(* CoDeSys 2.3.9.41 project: plc_110_main.pro *)
(* Libraries: D:\Projects\LittleProjects\Physical\Apartments\Slavutich2\SmartHouse\CoDeSys\lib\Timer.lib 12.1.22 22:29:23, STANDARD.LIB 4.10.05 11:14:46, IECSFC.LIB 13.4.06 15:51:28, C:\Program Files (x86)\Common Files\CAA-Targets\3S\Lib_PLCWinNT\SysLibCallback.lib 26.9.08 16:43:52, ANALYZATION.LIB 5.10.99 09:05:06 *)

(* PLC configuration (modules and I/O channels)
U1_FDI1_dimmer_button AT %IX0.0 [BitInput] FDI1_dimmer_button {ChannellName = Enter name}
U1_FDI2_dimmer_up AT %IX0.1 [BitInput] FDI2_dimmer_up {ChannellName = Enter name}
U1_FDI3_dimmer_down AT %IX0.2 [BitInput] FDI3_dimmer_down {ChannellName = Enter name}
U1_FDI4_NC AT %IX0.3 [BitInput] FDI4_NC {ChannellName = Enter name}
AT %IB1.0 [ByteInput] 8 discrete inputs {ChannellName = Enter name}
AT %IB1.1 [ByteInput] 8 discrete inputs {ChannellName = Enter name}
AT %IB1.2 [ByteInput] 8 discrete inputs {ChannellName = Enter name}
AT %IB1.3 [ByteInput] 8 discrete inputs {ChannellName = Enter name}
U1_DO1_warm_floor_room AT %QX2.0 [BitOutput] DO1_warm_floor_room {ChannellName = Enter name}
U1_DO2_warm_floor_logia AT %QX2.1 [BitOutput] DO2_warm_floor_logia {ChannellName = Enter name}
U1_DO3_warm_floor_kitchen AT %QX2.2 [BitOutput] DO3_warm_floor_kitchen {ChannellName = Enter name}
U1_DO4_warm_floor_hall AT %QX2.3 [BitOutput] DO4_warm_floor_hall {ChannellName = Enter name}
AT %QB3.0 [ByteOutput] 8 discrete outputs {ChannellName = Enter name}
AT %QB3.1 [ByteOutput] 8 discrete outputs {ChannellName = Enter name}
AT %QB3.2 [ByteOutput] 4 discrete outputs {ChannellName = Enter name}
Special input [ID103] node 4, in %IB4 out %QB4 {ChannellName = Special input}
  AT %IX4.0 [BitInput] Special input {ChannellName = Enter name}
Special output [ID104] node 5, in %IB5 out %QB5 {ChannellName = Special output}
  U1_PLC_speaker AT %QX5.0 [BitOutput] PLC_speaker {ChannellName = Enter name}
AT %QD6.0 [DWordOutput] Last address {ChannellName = Enter name}
AT %QW6.1 [WordOutput] Last error {ChannellName = Enter name}
RS-485-1 [COM1_USART] node 0, in %IB6.0 out %QB6.0 {ChannellName = RS-485-1; CommunicationSpeed = 115200; Parity = NO PARITY CHECK; BitLength = 8 bits; StopLength = One stop bit; InterfaceType = RS485; FrameOriented = RTU; Timeout = 0; Visibility = No}
Universal Modbus device [ID2000] node 1, in %IB6.1 out %QB6.1 {ChannellName = M1; ModuleIP = 10:0:0:223; ServiceTimeout = 150; TCPport = 502; NetMode = Serial; ModuleSlaveAddress = 1; RequestType = Both; PeriodOfService = 1000; Visibility = No; RepeatCounter = 0; ByteSequence = Trace_mode}
  AT %QB6.1.0 [ComChannel] Command (0xff - Start) {ChannellName = Enter name}
M1_DO1_door_lock_on AT %QW6.1.0.0 [WordOutput] {ChannellName = Enter name}
M1_DO2_doorbell_on AT %QW6.1.1.0 [WordOutput] {ChannellName = Enter name}
M1_DO3_door_lock_open_close AT %QW6.1.2.0 [WordOutput] {ChannellName = Enter name}
M1_DO4_cold_water_valve_close AT %QW6.1.3.0 [WordOutput] {ChannellName = Enter name}
M1_DO5_hot_water_valve_close AT %QW6.1.4.0 [WordOutput] {ChannellName = Enter name}
M1_DO6_water_valves_on AT %QW6.1.5.0 [WordOutput] {ChannellName = Enter name}
M1_DO7_NC AT %QW6.1.6.0 [WordOutput] {ChannellName = Enter name}
M1_DO8_siren_on AT %QW6.1.7.0 [WordOutput] {ChannellName = Enter name}
M1_DO_state AT %QW6.1.8.0 [WordOutput] {ChannellName = Enter name}
Universal Modbus device [ID2000] node 2, in %IB6.2 out %QB6.2 {ChannellName = Universal Modbus device; ModuleIP = 10:0:0:223; ServiceTimeout = 150; TCPport = 502; NetMode = Serial; ModuleSlaveAddress = 2; RequestType = Both; PeriodOfService = 1000; Visibility = No; RepeatCounter = 0; ByteSequence = Trace_mode}
  AT %QB6.2.0 [ComChannel] Command (0xff - Start) {ChannellName = Enter name}
M2_DO1_room_jalousie_up_down AT %QW6.2.0.0 [WordOutput] {ChannellName = Enter name}
M2_DO2_room_jalousie_on AT %QW6.2.1.0 [WordOutput] {ChannellName = Enter name}
M2_DO3_logia_jalousie_up_down AT %QW6.2.2.0 [WordOutput] {ChannellName = Enter name}
M2_DO4_logia_jalousie_on AT %QW6.2.3.0 [WordOutput] {ChannellName = Enter name}
M2_DO5_batroom_ventilation_fast_slow AT %QW6.2.4.0 [WordOutput] {ChannellName = Enter name}
M2_DO6_batroom_ventilation_on AT %QW6.2.5.0 [WordOutput] {ChannellName = Enter name}
M2_DO7_room_ventilation_fast_slow AT %QW6.2.6.0 [WordOutput] {ChannellName = Enter name}
M2_DO8_room_ventilation_on AT %QW6.2.7.0 [WordOutput] {ChannellName = Enter name}
M2_DO_state AT %QW6.2.8.0 [WordOutput] {ChannellName = Enter name}
AT %QB6.3.0 [ComChannel] Command (0xff - Start) {ChannellName = Enter name}
M3_IN1_status_warm_floor_room AT %QW6.3.0.0 [WordOutput] {ChannellName = Enter name}
M3_IN1_time_warm_floor_room AT %QW6.3.1.0 [WordOutput] {ChannellName = Enter name}
M3_IN1_temper_warm_floor_room AT %QD6.3.2.0 [FloatOutput] {ChannellName = Enter name}
M3_IN2_status_warm_floor_logia AT %QW6.3.3.0 [WordOutput] {ChannellName = Enter name}
M3_IN2_time_warm_floor_logia AT %QW6.3.4.0 [WordOutput] {ChannellName = Enter name}
M3_IN2_temper_warm_floor_logia AT %QD6.3.5.0 [FloatOutput] {ChannellName = Enter name}
M3_IN3_status_warm_floor_kitchen AT %QW6.3.6.0 [WordOutput] {ChannellName = Enter name}
M3_IN3_time_warm_floor_kitchen AT %QW6.3.7.0 [WordOutput] {ChannellName = Enter name}
M3_IN3_temper_warm_floor_kitchen AT %QD6.3.8.0 [FloatOutput] {ChannellName = Enter name}
M3_IN4_status_warm_floor_hall AT %QW6.3.9.0 [WordOutput] {ChannellName = Enter name}
M3_IN4_time_warm_floor_hall AT %QW6.3.10.0 [WordOutput] {ChannellName = Enter name}
M3_IN4_temper_warm_floor_hall AT %QD6.3.11.0 [FloatOutput] {ChannellName = Enter name}
M3_IN5_status_warm_floor_bathroom AT %QW6.3.12.0 [WordOutput] {ChannellName = Enter name}
M3_IN5_time_warm_floor_bathroom AT %QW6.3.13.0 [WordOutput] {ChannellName = Enter name}
M3_IN5_temper_warm_floor_bathroom AT %QD6.3.14.0 [FloatOutput] {ChannellName = Enter name}
M3_IN6_status_outdoor AT %QW6.3.15.0 [WordOutput] {ChannellName = Enter name}
ID2003NoNoINTRegister input module AT %QW6.3.16.0 [WordOutput] B%QB%MB%MM3_IN6_time_outdoor {ChannellName = Enter name}
M3_IN6_temper_outdoor AT %QD6.3.17.0 [FloatOutput] {ChannellName = Enter name}
M3_IN7_status_box AT %QW6.3.18.0 [WordOutput] {ChannellName = Enter name}
M3_IN7_time_box AT %QW6.3.19.0 [WordOutput] {ChannellName = Enter name}
M3_IN7_temper_box AT %QD6.3.20.0 [FloatOutput] {ChannellName = Enter name}
M3_IN8_status_luminosity_room AT %QW6.3.21.0 [WordOutput] {ChannellName = Enter name}
M3_IN8_time_luminosity_room AT %QW6.3.22.0 [WordOutput] {ChannellName = Enter name}
M3_IN8_luminosity_room AT %QD6.3.46.0 [FloatOutput] {ChannellName = Enter name}
AT %QB6.4.0 [ComChannel] Command (0xff - Start) {ChannellName = Enter name}
M4_AO1_room_converter_speed AT %QW6.4.0.0 [WordOutput] {ChannellName = Enter name}
M4_AO2_logia_converter_speed AT %QW6.4.1.0 [WordOutput] {ChannellName = Enter name}
M4_AO_3_NC AT %QW6.4.2.0 [WordOutput] {ChannellName = Enter name}
M4_AO_4_NC AT %QW6.4.3.0 [WordOutput] {ChannellName = Enter name}
M4_AO_5_NC AT %QW6.4.4.0 [WordOutput] {ChannellName = Enter name}
M4_AO_6_NC AT %QW6.4.5.0 [WordOutput] {ChannellName = Enter name}
AT %QB6.5.0 [ComChannel] Command (0xff - Start) {ChannellName = Enter name}
M5_AO1_room_light_1 AT %QW6.5.0.0 [WordOutput] {ChannellName = Enter name}
M5_AO2_room_light_2 AT %QW6.5.1.0 [WordOutput] {ChannellName = Enter name}
M5_AO3_logia_light AT %QW6.5.2.0 [WordOutput] {ChannellName = Enter name}
M5_AO4_kitchen_light AT %QW6.5.3.0 [WordOutput] {ChannellName = Enter name}
M5_AO5_hall_light AT %QW6.5.4.0 [WordOutput] {ChannellName = Enter name}
M5_AO6_bathroom_light AT %QW6.5.5.0 [WordOutput] {ChannellName = Enter name}
TCP [TCP_ID221] node 0, in %IB7.0.0 out %QB7.0.0 {ChannellName = TCP; RemotePort = 502; Visibility = No}
8 bits [8Bit] node 1, in %IB7.1 out %QB7.1 {ChannellName = 8 bit}
  AT %QB7.1.0 [ByteOutput] {ChannellName = Enter name}
8 bits [8Bit] node 2, in %IB7.2 out %QB7.2 {ChannellName = 8 bit}
  AT %QB7.2.0 [ByteOutput] {ChannellName = Enter name}
  AT %QB7.3.0 [ByteOutput] {ChannellName = Enter name}
  AT %QB7.4.0 [ByteOutput] {ChannellName = Enter name}
U1_R_002_room_light_intensity_1 AT %QW7.5.0 [WordOutput] {ChannellName = Enter name}
U1_R_003_room_light_intensity_2 AT %QW7.6.0 [WordOutput] {ChannellName = Enter name}
U1_R_004_logia_light_intensity AT %QW7.7.0 [WordOutput] {ChannellName = Enter name}
U1_R_005_kitchen_light_intensity AT %QW7.8.0 [WordOutput] {ChannellName = Enter name}
U1_R_006_hall_light_intensity AT %QW7.9.0 [WordOutput] {ChannellName = Enter name}
U1_R_007_bathroom_light_intensity AT %QW7.10.0 [WordOutput] {ChannellName = Enter name}
U1_R_008_room_light_change_rate AT %QW7.11.0 [WordOutput] {ChannellName = Enter name}
U1_R_009_other_light_change_rate AT %QW7.12.0 [WordOutput] {ChannellName = Enter name}
U1_R_010_room_light_correction_in_auto AT %QW7.13.0 [WordOutput] {ChannellName = Enter name}
*)

(* Task configuration *)
TASK U1_FDI1_dimmer_button (PRIORITY := 1, SINGLE := U1_FDI1_dimmer_button);
	DIMMER_HANDLER(act:=1);
END_TASK
TASK U1_FDI2_dimmer_up (PRIORITY := 1, SINGLE := U1_FDI2_dimmer_up);
	DIMMER_HANDLER(act:=2);
END_TASK
TASK FDI3_dimmer_down (PRIORITY := 1, SINGLE := U1_FDI3_dimmer_down);
	DIMMER_HANDLER(act:=3);
END_TASK
TASK dimmer_handler_tick (PRIORITY := 1, INTERVAL := T#100ms);
	DIMMER_HANDLER(act:=0);
END_TASK
TASK switch_handler_tick (PRIORITY := 1, INTERVAL := T#50ms);
	SWITCH_HANDLER();
END_TASK
TASK light_driver_tick (PRIORITY := 1, INTERVAL := T#40ms);
	LIGHT_DRIVER();
END_TASK
TASK light_auto_control_tick (PRIORITY := 1, INTERVAL := T#100ms);
	LIGHT_AUTO_CONTROL();
END_TASK

(* Global variable list: Global_Variables *)
VAR_GLOBAL
    PLC_STATUS: INT := 0;
END_VAR
VAR_GLOBAL CONSTANT
	PLC_RUN: INT := 2;
END_VAR

(* POU DIMMER_HANDLER, ST *)
PROGRAM DIMMER_HANDLER
VAR_INPUT
    act: INT; (* Action: 0 - tick (each 100 mills), 1 - U1_FDI1_dimmer_button, 2 - U1_FDI2_dimmer_up, 3 - FDI3_dimmer_down *)
END_VAR

VAR CONSTANT
    (* Input actions *)
    TICK: INT := 0;
    DIMMER_BUTTON: INT := 1;
    DIMMER_UP: INT := 2;
    DIMMER_DOWN: INT := 3;

    (* Parameters *)
    INDICATOR_BLINCK_TIME: INT := 3; (* 300 mills *)
    NUM_BLINCK_TO_SWITCH_MODE: INT := 4;  (* (300 * 4 * 2)mills *)
    DIMMER_RESET_TIME: INT := 100; (* 10 seconds *)
    DIMMING_STEP: INT := 10;
    DIMMING_MAX_VALUE: INT := 1000;
    ROOM_LIGHT_CHANGE_RATE: INT := 2;
    OTHER_LIGHT_CHANGE_RATE: INT := 5;
END_VAR

VAR
    dimmer_swith_count: INT := -1;
    dimmer_reset_count: INT := 0;
    is_room_dimmer: BOOL := TRUE;
    count: INT := 0;
END_VAR
(*
    Handeling of dimmer control handle

    Author: CAB 
    Cseated: 2022.01.25
*)

IF PLC_STATUS = PLC_RUN THEN
    IF act = TICK THEN
        IF U1_FDI1_dimmer_button AND dimmer_swith_count < (INDICATOR_BLINCK_TIME * NUM_BLINCK_TO_SWITCH_MODE * 2) AND dimmer_swith_count >= 0 THEN
            (* Count until switch dimmer mode room/other *)
            U1_DO12_dimer_mode_indication := ((dimmer_swith_count / INDICATOR_BLINCK_TIME) MOD 2) = BOOL_TO_INT(NOT is_room_dimmer);
            dimmer_swith_count := dimmer_swith_count + 1;

        ELSIF U1_FDI1_dimmer_button AND dimmer_swith_count > 0 THEN
            (* Do switch dimmer mode room/other   *)
            is_room_dimmer := NOT is_room_dimmer;
            U1_DO12_dimer_mode_indication := NOT is_room_dimmer;
            dimmer_swith_count := -1;

        ELSIF (NOT U1_FDI1_dimmer_button) AND dimmer_swith_count > 0 THEN
            (* Set mode indicator in case dimmer button is off before mode switched*)
            U1_DO12_dimer_mode_indication := NOT is_room_dimmer;
            dimmer_swith_count := -1;
        END_IF

        IF NOT is_room_dimmer THEN
            IF dimmer_reset_count >= DIMMER_RESET_TIME THEN
                is_room_dimmer := TRUE;
                U1_DO12_dimer_mode_indication := FALSE;
            END_IF
            dimmer_reset_count := dimmer_reset_count + 1;
        END_IF

    ELSIF act = DIMMER_BUTTON THEN
        U1_DO12_dimer_mode_indication := is_room_dimmer;
        dimmer_swith_count := 0;
        dimmer_reset_count := 0;
        U1_C_024_room_light_auto := FALSE; (* Reset light auto controll *)

    ELSIF act = DIMMER_UP THEN
        IF U1_FDI3_dimmer_down THEN
            IF is_room_dimmer AND NOT U1_C_024_room_light_auto THEN
                (* Decrising of room dimmers *)

                IF U1_C_016_room_light_1_on OR U1_C_017_room_light_2_on THEN
                    U1_R_008_room_light_change_rate := ROOM_LIGHT_CHANGE_RATE;
                END_IF

                IF U1_C_016_room_light_1_on AND U1_R_002_room_light_intensity_1 > DIMMING_STEP THEN
                    U1_R_002_room_light_intensity_1 := U1_R_002_room_light_intensity_1 - DIMMING_STEP;
                ELSIF U1_C_016_room_light_1_on THEN
                    U1_R_002_room_light_intensity_1 := 0;
                END_IF

                IF U1_C_017_room_light_2_on AND U1_R_003_room_light_intensity_2 > DIMMING_STEP THEN
                    U1_R_003_room_light_intensity_2 := U1_R_003_room_light_intensity_2 - DIMMING_STEP;
                ELSIF U1_C_017_room_light_2_on THEN
                    U1_R_003_room_light_intensity_2 := 0;
                END_IF

                U1_C_001_state_updated := TRUE;

            ELSIF NOT is_room_dimmer THEN
                (* Decrising of room other *)

                IF U1_C_018_logia_light_on OR U1_C_019_kitchen_light_on OR U1_C_020_hall_light_on OR U1_C_021_bathroom_light_on THEN
                    U1_R_009_other_light_change_rate := OTHER_LIGHT_CHANGE_RATE;
                END_IF

                IF U1_C_018_logia_light_on AND U1_R_004_logia_light_intensity > DIMMING_STEP THEN
                    U1_R_004_logia_light_intensity := U1_R_004_logia_light_intensity - DIMMING_STEP;
                ELSIF U1_C_018_logia_light_on THEN
                    U1_R_004_logia_light_intensity := 0;
                END_IF

                IF U1_C_019_kitchen_light_on AND U1_R_005_kitchen_light_intensity > DIMMING_STEP THEN
                    U1_R_005_kitchen_light_intensity := U1_R_005_kitchen_light_intensity - DIMMING_STEP;
                ELSIF U1_C_019_kitchen_light_on THEN
                    U1_R_005_kitchen_light_intensity := 0;
                END_IF

                IF U1_C_020_hall_light_on AND U1_R_006_hall_light_intensity > DIMMING_STEP THEN
                    U1_R_006_hall_light_intensity := U1_R_006_hall_light_intensity - DIMMING_STEP;
                ELSIF U1_C_020_hall_light_on THEN
                    U1_R_006_hall_light_intensity := 0;
                END_IF

                IF U1_C_021_bathroom_light_on AND U1_R_007_bathroom_light_intensity > DIMMING_STEP THEN
                    U1_R_007_bathroom_light_intensity := U1_R_007_bathroom_light_intensity - DIMMING_STEP;
                ELSIF U1_C_021_bathroom_light_on THEN
                    U1_R_007_bathroom_light_intensity := 0;
                END_IF

                U1_C_001_state_updated := TRUE;
            END_IF

            dimmer_reset_count := 0;
        END_IF

    ELSIF act = DIMMER_DOWN THEN
        IF U1_FDI2_dimmer_up THEN
            IF is_room_dimmer AND NOT U1_C_024_room_light_auto THEN
                (* Incrising of room dimmers *)

                IF U1_C_016_room_light_1_on OR U1_C_017_room_light_2_on THEN
                    U1_R_008_room_light_change_rate := ROOM_LIGHT_CHANGE_RATE;
                END_IF

                IF U1_C_016_room_light_1_on THEN
                    U1_R_002_room_light_intensity_1 := U1_R_002_room_light_intensity_1 + DIMMING_STEP;
                    IF U1_R_002_room_light_intensity_1 > DIMMING_MAX_VALUE THEN
                        U1_R_002_room_light_intensity_1 := DIMMING_MAX_VALUE;
                    END_IF
                END_IF

                IF U1_C_017_room_light_2_on THEN
                    U1_R_003_room_light_intensity_2 := U1_R_003_room_light_intensity_2 + DIMMING_STEP;
                    IF U1_R_003_room_light_intensity_2 > DIMMING_MAX_VALUE THEN
                        U1_R_003_room_light_intensity_2 := DIMMING_MAX_VALUE;
                    END_IF
                END_IF

                U1_C_001_state_updated := TRUE;

            ELSIF NOT is_room_dimmer THEN
                (* Incrising of room other *)

                IF U1_C_018_logia_light_on OR U1_C_019_kitchen_light_on OR U1_C_020_hall_light_on OR U1_C_021_bathroom_light_on THEN
                    U1_R_009_other_light_change_rate := OTHER_LIGHT_CHANGE_RATE;
                END_IF

                IF U1_C_018_logia_light_on THEN
                    U1_R_004_logia_light_intensity := U1_R_004_logia_light_intensity + DIMMING_STEP;
                    IF U1_R_004_logia_light_intensity > DIMMING_MAX_VALUE THEN
                        U1_R_004_logia_light_intensity := DIMMING_MAX_VALUE;
                    END_IF
                END_IF

                IF U1_C_019_kitchen_light_on THEN
                    U1_R_005_kitchen_light_intensity := U1_R_005_kitchen_light_intensity + DIMMING_STEP;
                    IF U1_R_005_kitchen_light_intensity > DIMMING_MAX_VALUE THEN
                        U1_R_005_kitchen_light_intensity := DIMMING_MAX_VALUE;
                    END_IF
                END_IF

                IF U1_C_020_hall_light_on THEN
                    U1_R_006_hall_light_intensity := U1_R_006_hall_light_intensity + DIMMING_STEP;
                    IF U1_R_006_hall_light_intensity > DIMMING_MAX_VALUE THEN
                        U1_R_006_hall_light_intensity := DIMMING_MAX_VALUE;
                    END_IF
                END_IF

                IF U1_C_021_bathroom_light_on THEN
                    U1_R_007_bathroom_light_intensity := U1_R_007_bathroom_light_intensity + DIMMING_STEP;
                    IF U1_R_007_bathroom_light_intensity > DIMMING_MAX_VALUE THEN
                        U1_R_007_bathroom_light_intensity := DIMMING_MAX_VALUE;
                    END_IF
                END_IF

                U1_C_001_state_updated := TRUE;
            END_IF

            dimmer_reset_count := 0;
        END_IF
    END_IF
END_IF
END_PROGRAM

(* POU SWITCH_HANDLER, ST *)
PROGRAM SWITCH_HANDLER
VAR
    hall_light_on: BOOL := FALSE;
    room_light_1: BOOL := FALSE;
    room_light_2: BOOL := FALSE;
    loggia_light: BOOL := FALSE;
    kitchen_light: BOOL := FALSE;
    bathroom_light: BOOL := FALSE;
    bathroom_ventilation: BOOL := FALSE;
    room_ventilation: BOOL := FALSE;
END_VAR
(*
    Handeling of switches over all rooms

    Author: CAB 
    Cseated: 2022.01.25
*)

IF PLC_STATUS = PLC_RUN THEN

    (* Handling of light switches *)
    
    IF (U1_DI5_pass_switch_light_room AND U1_DI10_pass_switch_light_hall) OR (NOT U1_DI5_pass_switch_light_room AND NOT U1_DI10_pass_switch_light_hall) THEN
        IF NOT hall_light_on THEN
            hall_light_on := TRUE;
            U1_C_020_hall_light_on := TRUE;
        END_IF
    ELSE
        IF hall_light_on THEN
            hall_light_on := FALSE;
            U1_C_020_hall_light_on := FALSE;
        END_IF
    END_IF

    IF U1_DI6_room_light_1 <> room_light_1 THEN
        room_light_1 := U1_DI6_room_light_1;
        U1_C_016_room_light_1_on := room_light_1;
    END_IF

    IF U1_DI7_room_light_2 <> room_light_2 THEN
        room_light_2 := U1_DI7_room_light_2;
        U1_C_017_room_light_2_on := room_light_2;
    END_IF

    IF U1_DI8_loggia_light <> loggia_light THEN
        loggia_light := U1_DI8_loggia_light;
        U1_C_018_logia_light_on := loggia_light;
    END_IF

    IF U1_DI9_kitchen_light <> kitchen_light THEN
        kitchen_light := U1_DI9_kitchen_light;
        U1_C_019_kitchen_light_on := kitchen_light;
    END_IF

    IF U1_DI11_bathroom_light <> bathroom_light THEN
        bathroom_light := U1_DI11_bathroom_light;
        U1_C_021_bathroom_light_on := bathroom_light;
    END_IF

    (* Handling of ventilation switches *)

    IF U1_DI12_bathroom_ventilation <> bathroom_ventilation THEN
        bathroom_ventilation := U1_DI12_bathroom_ventilation;
        (* TODO: Process it *)
    END_IF

    IF U1_DI17_room_ventilation <> room_ventilation THEN
        room_ventilation := U1_DI17_room_ventilation;
        (* TODO: Process it *)
    END_IF

END_IF
END_PROGRAM

(* POU LIGHT_DRIVER, ST *)
PROGRAM LIGHT_DRIVER
VAR CONSTANT
    (* Timeouts *)
    POWER_OFF_TIMEOUT: INT := 100; (* 40 * 100 = 4 second*)

    (* Input  bounds *)
    INTENCITY_MAX: INT := 1000;
    INTENCITY_MIN: INT := 0;

    (* Output  bounds *)
    OUT_MAX: INT := 1000; (* Max value alloved on output module*)
    ROOM_MAX_1: INT := 900;
    ROOM_MIN_1: INT := 100;
    ROOM_MAX_2: INT := 900;
    ROOM_MIN_2: INT := 100;
    ROOM_LOGIA_MAX: INT := 900;
    ROOM_LOGIA_MIN: INT := 100;
    ROOM_KITCHEN_MAX: INT := 900;
    ROOM_KITCHEN_MIN: INT := 100;
    ROOM_HALL_MAX: INT := 900;
    ROOM_HALL_MIN: INT := 100;
    ROOM_BATHROOM_MAX: INT := 900;
    ROOM_BATHROOM_MIN: INT := 100;
END_VAR
VAR
    (* Time counters *)
    room_light_off_counter: INT := 0;
    kitchen_off_counter: INT := 0;
    hall_off_counter: INT := 0;

    (* Normalized input *)
	room_light_intensity_1: INT := 0;
	room_light_intensity_2: INT := 0;
	logia_light_intensity: INT := 0;
	kitchen_light_intensity: INT := 0;
	hall_light_intensity: INT := 0;
	bathroom_light_intensity: INT := 0;
	room_light_change_rate: INT := 0;
	other_light_change_rate: INT := 0;

    (* Output *)
	room_light_out_1: INT := 0;
	room_light_out_2: INT := 0;
	logia_light_out: INT := 0;
	kitchen_light_out: INT := 0;
	hall_light_out: INT := 0;
	bathroom_light_out: INT := 0;

    (* Vars *)
    is_on: BOOL := FALSE;
    dif: INT := 0;
    change: INT := 0;
    scaled: INT := 0;
END_VAR
(*
    Control of LED light drivers

    Author: CAB 
    Cseated: 2022.01.25
    Called with 40ms timeout.
*)

IF PLC_STATUS = PLC_RUN THEN

    (* Set variables *)

    room_light_intensity_1 := U1_R_002_room_light_intensity_1;
    IF room_light_intensity_1 > INTENCITY_MAX THEN
        room_light_intensity_1 := INTENCITY_MAX;
    ELSIF room_light_intensity_1 < INTENCITY_MIN THEN
        room_light_intensity_1 := INTENCITY_MIN;
    END_IF

	room_light_intensity_2 := U1_R_003_room_light_intensity_2;
    IF room_light_intensity_2 > INTENCITY_MAX THEN
        room_light_intensity_2 := INTENCITY_MAX;
    ELSIF room_light_intensity_2 < INTENCITY_MIN THEN
        room_light_intensity_2 := INTENCITY_MIN;
    END_IF

	logia_light_intensity := U1_R_004_logia_light_intensity;
    IF logia_light_intensity > INTENCITY_MAX THEN
        logia_light_intensity := INTENCITY_MAX;
    ELSIF logia_light_intensity < INTENCITY_MIN THEN
        logia_light_intensity := INTENCITY_MIN;
    END_IF

	kitchen_light_intensity := U1_R_005_kitchen_light_intensity;
    IF kitchen_light_intensity > INTENCITY_MAX THEN
        kitchen_light_intensity := INTENCITY_MAX;
    ELSIF kitchen_light_intensity < INTENCITY_MIN THEN
        kitchen_light_intensity := INTENCITY_MIN;
    END_IF

	hall_light_intensity := U1_R_006_hall_light_intensity;
    IF hall_light_intensity > INTENCITY_MAX THEN
        hall_light_intensity := INTENCITY_MAX;
    ELSIF hall_light_intensity < INTENCITY_MIN THEN
        hall_light_intensity := INTENCITY_MIN;
    END_IF

	bathroom_light_intensity := U1_R_007_bathroom_light_intensity;
    IF bathroom_light_intensity > INTENCITY_MAX THEN
        bathroom_light_intensity := INTENCITY_MAX;
    ELSIF bathroom_light_intensity < INTENCITY_MIN THEN
        bathroom_light_intensity := INTENCITY_MIN;
    END_IF

    room_light_change_rate := U1_R_008_room_light_change_rate;
    IF room_light_change_rate > INTENCITY_MAX THEN
        room_light_change_rate := INTENCITY_MAX;
    ELSIF room_light_change_rate < INTENCITY_MIN THEN
        room_light_change_rate := INTENCITY_MIN;
    END_IF

    other_light_change_rate := U1_R_009_other_light_change_rate;
    IF other_light_change_rate > INTENCITY_MAX THEN
        other_light_change_rate := INTENCITY_MAX;
    ELSIF other_light_change_rate < INTENCITY_MIN THEN
        other_light_change_rate := INTENCITY_MIN;
    END_IF

    (* On/off power relay *)

    is_on := U1_C_016_room_light_1_on OR U1_C_017_room_light_2_on OR room_light_out_1 > INTENCITY_MIN OR room_light_out_2 > INTENCITY_MIN;
    IF is_on AND (NOT U1_DO9_room_light_power) THEN
        U1_DO9_room_light_power := TRUE;
        room_light_off_counter := POWER_OFF_TIMEOUT;
    ELSIF NOT is_on THEN
        IF room_light_off_counter <= 0 AND U1_DO9_room_light_power THEN
            U1_DO9_room_light_power := FALSE;
        ELSIF room_light_off_counter > 0 THEN
            room_light_off_counter := room_light_off_counter - 1;
        END_IF
    ELSE
        room_light_off_counter := POWER_OFF_TIMEOUT;
    END_IF

    is_on := U1_C_018_logia_light_on OR U1_C_019_kitchen_light_on OR logia_light_out > INTENCITY_MIN OR kitchen_light_out > INTENCITY_MIN;
    IF is_on AND (NOT U1_DO10_logia_kitchen_light_power) THEN
        U1_DO10_logia_kitchen_light_power := TRUE;
        kitchen_off_counter := POWER_OFF_TIMEOUT;
    ELSIF NOT is_on THEN
        IF kitchen_off_counter <= 0 AND U1_DO10_logia_kitchen_light_power THEN
            U1_DO10_logia_kitchen_light_power := FALSE;
        ELSIF kitchen_off_counter > 0 THEN
            kitchen_off_counter := kitchen_off_counter - 1;
        END_IF
    ELSE
        kitchen_off_counter := POWER_OFF_TIMEOUT;
    END_IF

    is_on := U1_C_020_hall_light_on OR U1_C_021_bathroom_light_on OR hall_light_out > INTENCITY_MIN OR bathroom_light_out > INTENCITY_MIN;
    IF is_on AND (NOT U1_DO11_hall_bathroom_light_power) THEN
        U1_DO11_hall_bathroom_light_power := TRUE;
        hall_off_counter := POWER_OFF_TIMEOUT;
    ELSIF NOT is_on THEN
        IF hall_off_counter <= 0 AND U1_DO11_hall_bathroom_light_power THEN
            U1_DO11_hall_bathroom_light_power := FALSE;
        ELSIF hall_off_counter > 0 THEN
            hall_off_counter := hall_off_counter - 1;
        END_IF
    ELSE
        hall_off_counter := POWER_OFF_TIMEOUT;
    END_IF

    (* Smooth light controll *)

    IF U1_C_016_room_light_1_on THEN
        dif := room_light_intensity_1 - room_light_out_1;
        IF dif <> 0 THEN
            IF ABS(dif) <= room_light_change_rate THEN
                change := dif;
            ELSE
                change := room_light_change_rate;
                IF dif < 0 THEN
                    change := change * -1;
                END_IF
            END_IF
            room_light_out_1 := room_light_out_1 + change;
        END_IF
    ELSIF room_light_out_1 > 0 THEN
       room_light_out_1 := room_light_out_1 - room_light_change_rate;
       IF room_light_out_1 < 0 THEN
           room_light_out_1 := 0;
       END_IF
    END_IF

    IF U1_C_017_room_light_2_on THEN
        dif := room_light_intensity_2 - room_light_out_2;
        IF dif <> 0 THEN
            IF ABS(dif) <= room_light_change_rate THEN
                change := dif;
            ELSE
                change := room_light_change_rate;
                IF dif < 0 THEN
                    change := change * -1;
                END_IF
            END_IF
            room_light_out_2 := room_light_out_2 + change;
        END_IF
    ELSIF room_light_out_2 > 0 THEN
       room_light_out_2 := room_light_out_2 - room_light_change_rate;
       IF room_light_out_2 < 0 THEN
           room_light_out_2 := 0;
       END_IF
    END_IF

    IF U1_C_018_logia_light_on THEN
        dif := logia_light_intensity - logia_light_out;
        IF dif <> 0 THEN
            IF ABS(dif) <= other_light_change_rate THEN
                change := dif;
            ELSE
                change := other_light_change_rate;
                IF dif < 0 THEN
                    change := change * -1;
                END_IF
            END_IF
            logia_light_out := logia_light_out + change;
        END_IF
    ELSIF logia_light_out > 0 THEN
       logia_light_out := logia_light_out - other_light_change_rate;
       IF logia_light_out < 0 THEN
           logia_light_out := 0;
       END_IF
    END_IF

    IF U1_C_019_kitchen_light_on THEN
        dif := kitchen_light_intensity - kitchen_light_out;
        IF dif <> 0 THEN
            IF ABS(dif) <= other_light_change_rate THEN
                change := dif;
            ELSE
                change := other_light_change_rate;
                IF dif < 0 THEN
                    change := change * -1;
                END_IF
            END_IF
            kitchen_light_out := kitchen_light_out + change;
        END_IF
    ELSIF kitchen_light_out > 0 THEN
       kitchen_light_out := kitchen_light_out - other_light_change_rate;
       IF kitchen_light_out < 0 THEN
           kitchen_light_out := 0;
       END_IF
    END_IF

    IF U1_C_020_hall_light_on THEN
        dif := hall_light_intensity - hall_light_out;
        IF dif <> 0 THEN
            IF ABS(dif) <= other_light_change_rate THEN
                change := dif;
            ELSE
                change := other_light_change_rate;
                IF dif < 0 THEN
                    change := change * -1;
                END_IF
            END_IF
            hall_light_out := hall_light_out + change;
        END_IF
    ELSIF hall_light_out > 0 THEN
       hall_light_out := hall_light_out - other_light_change_rate;
       IF hall_light_out < 0 THEN
           hall_light_out := 0;
       END_IF
    END_IF

    IF U1_C_021_bathroom_light_on THEN
        dif := bathroom_light_intensity - bathroom_light_out;
        IF dif <> 0 THEN
            IF ABS(dif) <= other_light_change_rate THEN
                change := dif;
            ELSE
                change := other_light_change_rate;
                IF dif < 0 THEN
                    change := change * -1;
                END_IF
            END_IF
            bathroom_light_out := bathroom_light_out + change;
        END_IF
    ELSIF bathroom_light_out > 0 THEN
       bathroom_light_out := bathroom_light_out - other_light_change_rate;
       IF bathroom_light_out < 0 THEN
           bathroom_light_out := 0;
       END_IF
    END_IF

    (* Ouutput scaling *)

    IF room_light_out_1 > 0 THEN
        scaled := ROOM_MIN_1 + REAL_TO_INT(INT_TO_REAL(room_light_out_1) * (INT_TO_REAL(ROOM_MAX_1 - ROOM_MIN_1) / OUT_MAX));
        IF scaled <> M5_AO1_room_light_1 THEN
            M5_AO1_room_light_1 := scaled;
        END_IF
    ELSIF M5_AO1_room_light_1 <> 0 THEN
        M5_AO1_room_light_1 := 0;
    END_IF

    IF room_light_out_2 > 0 THEN
        scaled := ROOM_MIN_2 + REAL_TO_INT(INT_TO_REAL(room_light_out_2) * (INT_TO_REAL(ROOM_MAX_2 - ROOM_MIN_2) / OUT_MAX));
        IF scaled <> M5_AO2_room_light_2 THEN
            M5_AO2_room_light_2 := scaled;
        END_IF
    ELSIF M5_AO2_room_light_2 <> 0 THEN
        M5_AO2_room_light_2 := 0;
    END_IF

    IF logia_light_out > 0 THEN
        scaled := ROOM_LOGIA_MIN + REAL_TO_INT(INT_TO_REAL(logia_light_out) * (INT_TO_REAL(ROOM_LOGIA_MAX - ROOM_LOGIA_MIN) / OUT_MAX));
        IF scaled <> M5_AO3_logia_light THEN
            M5_AO3_logia_light := scaled;
        END_IF
    ELSIF M5_AO3_logia_light <> 0 THEN
        M5_AO3_logia_light := 0;
    END_IF

    IF kitchen_light_out > 0 THEN
        scaled := ROOM_KITCHEN_MIN + REAL_TO_INT(INT_TO_REAL(kitchen_light_out) * (INT_TO_REAL(ROOM_KITCHEN_MAX - ROOM_KITCHEN_MIN) / OUT_MAX));
        IF scaled <> M5_AO4_kitchen_light THEN
            M5_AO4_kitchen_light := scaled;
        END_IF
    ELSIF M5_AO4_kitchen_light <> 0 THEN
        M5_AO4_kitchen_light := 0;
    END_IF

    IF hall_light_out > 0 THEN
        scaled := ROOM_HALL_MIN + REAL_TO_INT(INT_TO_REAL(hall_light_out) * (INT_TO_REAL(ROOM_HALL_MAX - ROOM_HALL_MIN) / OUT_MAX));
        IF scaled <> M5_AO5_hall_light THEN
            M5_AO5_hall_light := scaled;
        END_IF
    ELSIF M5_AO5_hall_light <> 0 THEN
        M5_AO5_hall_light := 0;
    END_IF

    IF bathroom_light_out > 0 THEN
        scaled := ROOM_BATHROOM_MIN + REAL_TO_INT(INT_TO_REAL(bathroom_light_out) * (INT_TO_REAL(ROOM_BATHROOM_MAX - ROOM_BATHROOM_MIN) / OUT_MAX));
        IF scaled <> M5_AO6_bathroom_light THEN
            M5_AO6_bathroom_light := scaled;
        END_IF
    ELSIF M5_AO6_bathroom_light <> 0 THEN
        M5_AO6_bathroom_light := 0;
    END_IF
END_IF
END_PROGRAM

(* POU LIGHT_AUTO_CONTROL, ST *)
PROGRAM LIGHT_AUTO_CONTROL
VAR CONSTANT
    MIN_INTENSITY_1: INT := 0;
	MAX_INTENSITY_1: INT := 1000;
    MIN_INTENSITY_2: INT := 0;
	MAX_INTENSITY_2: INT := 1000;
    SENSORE_SCALING: REAL := 1.0;
    EFFECT_PROPORTION: REAL := 0.1;
END_VAR
VAR
    effect: INT := 0;
END_VAR
(*
    Automatic control of the light intensity in room

    Author: CAB 
    Cseated: 2022.02.07
*)

IF PLC_STATUS = PLC_RUN AND U1_C_024_room_light_auto AND (U1_C_016_room_light_1_on OR U1_C_017_room_light_2_on) AND M3_IN8_status_luminosity_room = 0 THEN

    (* Calculate effect *)

    effect := REAL_TO_INT(WORD_TO_REAL(U1_R_010_room_light_correction_in_auto) - (M3_IN8_luminosity_room * SENSORE_SCALING));

    (* Change light intensity *)

    IF U1_C_016_room_light_1_on THEN
        U1_R_002_room_light_intensity_1 := U1_R_002_room_light_intensity_1 + effect;
        IF U1_R_002_room_light_intensity_1 < MIN_INTENSITY_1 THEN
            U1_R_002_room_light_intensity_1 := MIN_INTENSITY_1;
        END_IF
        IF U1_R_002_room_light_intensity_1 > MAX_INTENSITY_1 THEN
            U1_R_002_room_light_intensity_1 := MAX_INTENSITY_1;
        END_IF
    END_IF

    IF U1_C_017_room_light_2_on THEN
        U1_R_003_room_light_intensity_2 := U1_R_003_room_light_intensity_2 + effect;

        IF U1_R_003_room_light_intensity_2 < MIN_INTENSITY_2 THEN
            U1_R_003_room_light_intensity_2 := MIN_INTENSITY_2;
        END_IF

        IF U1_R_003_room_light_intensity_2 < MIN_INTENSITY_2 THEN
            U1_R_003_room_light_intensity_2 := MIN_INTENSITY_2;
        END_IF

    END_IF

ELSIF M3_IN8_status_luminosity_room <> 0 THEN

    (* Set error flag in case sensore failed *)

    U1_C_025_light_error := TRUE;

END_IF
END_PROGRAM

(* POU PLC_PRG, ST *)
PROGRAM PLC_PRG
VAR

END_VAR
(*
    Main program

    Author: CAB 
    Cseated: 2022.01.25
*)

PLC_STATUS := PLC_RUN;  (* TODO: To implement starting process *)
END_PROGRAM

(* POU START, ST *)
FUNCTION START: DWORD
VAR_INPUT
	dwEvent: INT;
	dwFilter: INT;
	dwOwner: INT;
END_VAR
(*
    Initialisation function

    Author: CAB 
    Cseated: 2022.01.25
*)

PLC_STATUS := PLC_RUN;  (* TODO: To implement starting process *)

U1_R_002_room_light_intensity_1 := 500;
U1_R_003_room_light_intensity_2 := 500;
U1_R_004_logia_light_intensity := 500;
U1_R_005_kitchen_light_intensity := 500;
U1_R_006_hall_light_intensity := 500;
U1_R_007_bathroom_light_intensity := 500;

U1_R_008_room_light_change_rate := 10;
U1_R_009_other_light_change_rate := 10;

U1_C_024_room_light_auto := FALSE;
U1_R_010_room_light_correction_in_auto := 0;

U1_DO1_warm_floor_room := TRUE;
END_FUNCTION
